(* IEC 61131-3 sources: plcc/tests/fixtures/programs, 8 files *)

(* ---- alarm_system.st ---- *)
FUNCTION PriorityEncode : INT
VAR_INPUT critical : INT; high : INT; medium : INT; low : INT; END_VAR
    IF critical <> 0 THEN PriorityEncode := 4;
    ELSIF high <> 0 THEN PriorityEncode := 3;
    ELSIF medium <> 0 THEN PriorityEncode := 2;
    ELSIF low <> 0 THEN PriorityEncode := 1;
    ELSE PriorityEncode := 0;
    END_IF;
END_FUNCTION

FUNCTION_BLOCK AlarmHandler
VAR_INPUT
    temp_alarm : BOOL;
    pressure_alarm : BOOL;
    level_alarm : BOOL;
END_VAR
VAR_OUTPUT
    alarm_active : BOOL;
    alarm_code : INT;
END_VAR
VAR
    temp_val : INT;
    press_val : INT;
    level_val : INT;
END_VAR
    IF temp_alarm THEN temp_val := 1; ELSE temp_val := 0; END_IF;
    IF pressure_alarm THEN press_val := 1; ELSE press_val := 0; END_IF;
    IF level_alarm THEN level_val := 1; ELSE level_val := 0; END_IF;
    alarm_code := PriorityEncode(press_val, temp_val, level_val, 0);
    alarm_active := alarm_code > 0;
END_FUNCTION_BLOCK

PROGRAM AlarmSystem
VAR
    handler : AlarmHandler;
    system_alarm : BOOL;
    system_code : INT;
END_VAR
    handler(temp_alarm := TRUE, pressure_alarm := FALSE, level_alarm := TRUE);
    system_alarm := handler.alarm_active;
    system_code := handler.alarm_code;
END_PROGRAM

(* ---- motor_control.st ---- *)
FUNCTION_BLOCK MotorController
VAR_INPUT
    start_cmd : BOOL;
    stop_cmd : BOOL;
    current : REAL;
    overload_limit : REAL := 15.0;
END_VAR
VAR_OUTPUT
    running : BOOL;
    fault : BOOL;
    run_time : INT;
END_VAR
VAR
    overload_count : INT := 0;
END_VAR
    IF stop_cmd OR fault THEN
        running := FALSE;
    ELSIF start_cmd AND NOT fault THEN
        running := TRUE;
    END_IF;

    IF running THEN
        run_time := run_time + 1;
        IF current > overload_limit THEN
            overload_count := overload_count + 1;
            IF overload_count >= 3 THEN
                fault := TRUE;
                running := FALSE;
            END_IF;
        ELSE
            overload_count := 0;
        END_IF;
    END_IF;
END_FUNCTION_BLOCK

PROGRAM MotorSystem
VAR
    motor1 : MotorController;
    motor2 : MotorController;
    any_fault : BOOL;
END_VAR
    motor1(start_cmd := TRUE, stop_cmd := FALSE, current := 10.0);
    motor2(start_cmd := TRUE, stop_cmd := FALSE, current := 10.0);
    any_fault := motor1.fault OR motor2.fault;
END_PROGRAM

(* ---- pid_simple.st ---- *)
FUNCTION_BLOCK PID
VAR_INPUT
    setpoint : REAL;
    measured : REAL;
    kp : REAL := 1.0;
    ki : REAL := 0.1;
    kd : REAL := 0.05;
    dt : REAL := 0.01;
    out_min : REAL := -100.0;
    out_max : REAL := 100.0;
END_VAR
VAR_OUTPUT
    output : REAL;
END_VAR
VAR
    err : REAL;
    prev_err : REAL := 0.0;
    integral : REAL := 0.0;
    derivative : REAL;
END_VAR
    err := setpoint - measured;
    integral := integral + err * dt;
    derivative := (err - prev_err) / dt;
    output := kp * err + ki * integral + kd * derivative;

    (* Clamp output *)
    IF output > out_max THEN
        output := out_max;
    ELSIF output < out_min THEN
        output := out_min;
    END_IF;

    prev_err := err;
END_FUNCTION_BLOCK

PROGRAM PIDController
VAR
    pid_inst : PID;
    sensor_value : REAL := 0.0;
    target_value : REAL := 50.0;
    control_output : REAL;
END_VAR
    pid_inst(setpoint := target_value, measured := sensor_value);
    control_output := pid_inst.output;
END_PROGRAM

(* ---- water_treatment.st ---- *)
(* Water Treatment Plant Control *)
(* Multiple tanks, pumps, valves, level/flow sensors *)
(* A realistic industrial PLC program with multiple FBs, *)
(* process control, alarm handling, and Modbus-mappable state. *)

FUNCTION_BLOCK TankLevel
VAR_INPUT
    inlet_flow : REAL;      (* L/min *)
    outlet_flow : REAL;     (* L/min *)
    max_capacity : REAL;    (* Liters *)
END_VAR
VAR_OUTPUT
    level : REAL;           (* Current level in Liters *)
    level_pct : INT;        (* 0-100% *)
    high_alarm : BOOL;
    low_alarm : BOOL;
END_VAR
VAR
    high_limit : REAL := 90.0;  (* % *)
    low_limit : REAL := 10.0;   (* % *)
END_VAR
    level := level + (inlet_flow - outlet_flow) * 0.001;  (* dt = 1ms sim *)
    IF level < 0.0 THEN level := 0.0; END_IF;
    IF level > max_capacity THEN level := max_capacity; END_IF;
    level_pct := REAL_TO_INT(level * 100.0 / max_capacity);
    high_alarm := level_pct > REAL_TO_INT(high_limit);
    low_alarm := level_pct < REAL_TO_INT(low_limit);
END_FUNCTION_BLOCK

FUNCTION_BLOCK PumpControl
VAR_INPUT
    enable : BOOL;
    speed_setpoint : INT;   (* 0-100% *)
    fault_reset : BOOL;
END_VAR
VAR_OUTPUT
    running : BOOL;
    actual_speed : INT;
    fault : BOOL;
    runtime_hrs : INT;
END_VAR
VAR
    runtime_scans : INT := 0;
END_VAR
    IF fault_reset THEN fault := FALSE; END_IF;
    IF enable AND NOT fault THEN
        running := TRUE;
        actual_speed := speed_setpoint;
        runtime_scans := runtime_scans + 1;
        runtime_hrs := runtime_scans / 3600;  (* assuming 1 scan/sec *)
    ELSE
        running := FALSE;
        actual_speed := 0;
    END_IF;
END_FUNCTION_BLOCK

FUNCTION_BLOCK ValveControl
VAR_INPUT
    open_cmd : BOOL;
    close_cmd : BOOL;
END_VAR
VAR_OUTPUT
    position : INT;   (* 0=closed, 100=open *)
    is_open : BOOL;
    is_closed : BOOL;
END_VAR
    IF open_cmd AND NOT close_cmd THEN
        IF position < 100 THEN position := position + 5; END_IF;
    ELSIF close_cmd AND NOT open_cmd THEN
        IF position > 0 THEN position := position - 5; END_IF;
    END_IF;
    is_open := position >= 100;
    is_closed := position <= 0;
END_FUNCTION_BLOCK

PROGRAM WaterTreatment
VAR
    (* Process state *)
    mode : INT := 0;        (* 0=stop, 1=run, 2=flush, 3=alarm *)
    cycle_count : INT := 0;

    (* Tanks *)
    raw_tank : TankLevel;
    clean_tank : TankLevel;

    (* Pumps *)
    inlet_pump : PumpControl;
    transfer_pump : PumpControl;
    outlet_pump : PumpControl;

    (* Valves *)
    inlet_valve : ValveControl;
    outlet_valve : ValveControl;
    drain_valve : ValveControl;

    (* Setpoints — these are Modbus-writable *)
    raw_tank_sp : INT := 50;     (* target level % *)
    clean_tank_sp : INT := 70;   (* target level % *)
    inlet_speed : INT := 60;     (* pump speed % *)
    transfer_speed : INT := 40;
    outlet_speed : INT := 30;

    (* Status — these are Modbus-readable *)
    system_ok : BOOL := TRUE;
    alarm_count : INT := 0;
    total_flow : INT := 0;
END_VAR
    cycle_count := cycle_count + 1;

    CASE mode OF
        0: (* STOPPED *)
            inlet_pump(enable := FALSE, speed_setpoint := 0, fault_reset := FALSE);
            transfer_pump(enable := FALSE, speed_setpoint := 0, fault_reset := FALSE);
            outlet_pump(enable := FALSE, speed_setpoint := 0, fault_reset := FALSE);
            inlet_valve(open_cmd := FALSE, close_cmd := TRUE);
            outlet_valve(open_cmd := FALSE, close_cmd := TRUE);
            drain_valve(open_cmd := FALSE, close_cmd := TRUE);

        1: (* RUNNING *)
            (* Control raw water tank level *)
            IF raw_tank.level_pct < raw_tank_sp THEN
                inlet_pump(enable := TRUE, speed_setpoint := inlet_speed, fault_reset := FALSE);
                inlet_valve(open_cmd := TRUE, close_cmd := FALSE);
            ELSE
                inlet_pump(enable := FALSE, speed_setpoint := 0, fault_reset := FALSE);
                inlet_valve(open_cmd := FALSE, close_cmd := TRUE);
            END_IF;

            (* Transfer from raw to clean *)
            IF raw_tank.level_pct > 20 AND clean_tank.level_pct < clean_tank_sp THEN
                transfer_pump(enable := TRUE, speed_setpoint := transfer_speed, fault_reset := FALSE);
            ELSE
                transfer_pump(enable := FALSE, speed_setpoint := 0, fault_reset := FALSE);
            END_IF;

            (* Outlet pump *)
            IF clean_tank.level_pct > 30 THEN
                outlet_pump(enable := TRUE, speed_setpoint := outlet_speed, fault_reset := FALSE);
                outlet_valve(open_cmd := TRUE, close_cmd := FALSE);
            ELSE
                outlet_pump(enable := FALSE, speed_setpoint := 0, fault_reset := FALSE);
                outlet_valve(open_cmd := FALSE, close_cmd := TRUE);
            END_IF;

            drain_valve(open_cmd := FALSE, close_cmd := TRUE);

        2: (* FLUSH *)
            inlet_pump(enable := FALSE, speed_setpoint := 0, fault_reset := FALSE);
            transfer_pump(enable := FALSE, speed_setpoint := 0, fault_reset := FALSE);
            outlet_pump(enable := FALSE, speed_setpoint := 0, fault_reset := FALSE);
            inlet_valve(open_cmd := FALSE, close_cmd := TRUE);
            outlet_valve(open_cmd := FALSE, close_cmd := TRUE);
            drain_valve(open_cmd := TRUE, close_cmd := FALSE);

        3: (* ALARM *)
            inlet_pump(enable := FALSE, speed_setpoint := 0, fault_reset := FALSE);
            transfer_pump(enable := FALSE, speed_setpoint := 0, fault_reset := FALSE);
            outlet_pump(enable := FALSE, speed_setpoint := 0, fault_reset := FALSE);
            inlet_valve(open_cmd := FALSE, close_cmd := TRUE);
            outlet_valve(open_cmd := FALSE, close_cmd := TRUE);
            drain_valve(open_cmd := FALSE, close_cmd := TRUE);
    END_CASE;

    (* Update tank levels *)
    raw_tank(
        inlet_flow := INT_TO_REAL(inlet_pump.actual_speed) * 0.5,
        outlet_flow := INT_TO_REAL(transfer_pump.actual_speed) * 0.3,
        max_capacity := 1000.0
    );
    clean_tank(
        inlet_flow := INT_TO_REAL(transfer_pump.actual_speed) * 0.3,
        outlet_flow := INT_TO_REAL(outlet_pump.actual_speed) * 0.2,
        max_capacity := 500.0
    );

    (* Alarm handling *)
    IF raw_tank.high_alarm OR clean_tank.high_alarm THEN
        alarm_count := alarm_count + 1;
        IF alarm_count > 100 THEN
            mode := 3;
            system_ok := FALSE;
        END_IF;
    ELSE
        alarm_count := 0;
    END_IF;

    total_flow := total_flow + outlet_pump.actual_speed;
END_PROGRAM

(* ---- batch_process.st ---- *)
PROGRAM BatchProcess
VAR
    stage : INT := 0;
    timer : INT := 0;
    fill_valve : BOOL := FALSE;
    mixer : BOOL := FALSE;
    drain_valve : BOOL := FALSE;
    batch_count : INT := 0;
    complete : BOOL := FALSE;
END_VAR
    timer := timer + 1;
    CASE stage OF
        0: (* IDLE *)
            fill_valve := FALSE; mixer := FALSE; drain_valve := FALSE;
            stage := 1; timer := 0;
        1: (* FILL *)
            fill_valve := TRUE;
            IF timer >= 20 THEN stage := 2; timer := 0; fill_valve := FALSE; END_IF;
        2: (* MIX *)
            mixer := TRUE;
            IF timer >= 30 THEN stage := 3; timer := 0; mixer := FALSE; END_IF;
        3: (* DRAIN *)
            drain_valve := TRUE;
            IF timer >= 15 THEN
                stage := 0; timer := 0; drain_valve := FALSE;
                batch_count := batch_count + 1;
                complete := TRUE;
            END_IF;
    ELSE
        stage := 0;
    END_CASE;
END_PROGRAM

(* ---- blink.st ---- *)
PROGRAM Blink
VAR
    output : BOOL := FALSE;
END_VAR
    output := NOT output;
END_PROGRAM

(* ---- state_machine.st ---- *)
PROGRAM StateMachine
VAR
    state : INT := 0;
    output_a : BOOL := FALSE;
    output_b : BOOL := FALSE;
    input_trigger : BOOL := FALSE;
    counter : INT := 0;
END_VAR
    CASE state OF
        0:
            output_a := FALSE;
            output_b := FALSE;
            IF input_trigger THEN
                state := 1;
            END_IF;
        1:
            output_a := TRUE;
            output_b := FALSE;
            counter := counter + 1;
            IF counter >= 10 THEN
                state := 2;
                counter := 0;
            END_IF;
        2:
            output_a := FALSE;
            output_b := TRUE;
            counter := counter + 1;
            IF counter >= 5 THEN
                state := 0;
                counter := 0;
            END_IF;
    ELSE
        state := 0;
    END_CASE;
END_PROGRAM

(* ---- stdlib_blinker.st ---- *)
(* SPDX-License-Identifier: MPL-2.0 *)
(*
 * A blinker built entirely from IEC 61131-3 standard function blocks.
 *
 * Requires the bundled ST standard library, i.e. the default
 * `--stdlib bundled-st`. With `--stdlib none` this fails to compile with an
 * "unknown type `TON`" diagnostic rather than silently doing nothing.
 *
 * The timers read the platform clock via `plcc_monotonic_ns`, so `on_time` and
 * `off_time` are real durations and do not drift with scan period.
 *)
PROGRAM StdlibBlinker
VAR
    (* One-shot rearm chain: on_delay expires -> lamp off, off_delay expires -> lamp on *)
    on_delay : TON;
    off_delay : TON;
    edge : R_TRIG;
    cycles : CTU;

    lamp : BOOL := TRUE;
    cycle_count : INT;
    reset_count : BOOL := FALSE;
END_VAR
    on_delay(IN := lamp, PT := T#250ms);
    IF on_delay.Q THEN
        lamp := FALSE;
    END_IF;

    off_delay(IN := NOT lamp, PT := T#250ms);
    IF off_delay.Q THEN
        lamp := TRUE;
    END_IF;

    (* Count completed off->on transitions of the lamp. *)
    edge(CLK := lamp);
    cycles(CU := edge.Q, R := reset_count, PV := 1000);
    cycle_count := cycles.CV;
END_PROGRAM
